# EPICS substitutions: epics/transprofs_tb.subs
file transprofs_tb.template {
  pattern { DEVICE}
  	  { "$(DEVICE)"}
}

file transprofs_wirescan.template {
  pattern { DEVICE}
  	  { "$(DEVICE)"}
}
